(* IEC 61131-3 sources: CodesysTest/alpha/export/Pro18_1174_HilscherCard.dev/Plc Logic/Application/Motors/Applied Motion/FB_AppliedMotionStepServoEIPBaseQX.pou, 1 file *)

(* ---- MoveDistanceTorque.m.st ---- *)
(*#-#-#-#-#-#-#-#-#-#---Declaration---#-#-#-#-#-#-#-#-#-#-#-#-#*)

METHOD MoveDistanceTorque
VAR_INPUT
	(*Distance to move in inches*)
    distance    : REAL;
    (*Acceleration in RPM/sec*)
    acceleration    : INT;
    (*Deceleration in RPM/sec*)
    deceleration    : INT;
    (*Velocity in .25RPM*)
    velocity    : INT;
	(*Current in .01A*)
	current : DINT;
END_VAR
(*#-#-#-#-#-#-#-#-#-#---Implementation---#-#-#-#-#-#-#-#-#-#-#-#-#*)

//This method preps the data to send to the drive and triggers the send.
//Set distance and unpack to prep data to send to motor

commandSuccessful := FALSE;

distanceToMoveInSteps := REAL_TO_DINT((distance) * stepsPerInchSetpoint);
IF reversePolarity THEN
    distanceToMoveInSteps := distanceToMoveInSteps * -1;
END_IF

pointToPointAccelSetpoint := acceleration;
pointToPointDecelSetpoint := deceleration;
velocitySetpoint := velocity;
currentLimit := current;

parameter1 := 2;
commands.SendQAndExecute := TRUE;
